FUNCTION_BLOCK "Syntax_MissingBegin"
{ S7_Optimized_Access := 'TRUE' }
VERSION : 0.1

VAR
    value : Int;
END_VAR

    #value := 1;
    // EXPECT: error[syntax.expected-begin] SYN-BLOCK-001
END_FUNCTION_BLOCK
